// TIA Portal V17 export
// export: Created 2023-05-07T12:12:23.0932555Z, ExportSetting WithDefaults, DisplayName Totally Integrated Automation Portal, DisplayVersion V17, DisplayName TIA Portal Openness, DisplayVersion V17, DisplayName TIA Portal Version Control Interface, DisplayVersion V17, DisplayName TIA Portal Test Suite Advanced, DisplayVersion V17, DisplayName STEP 7 Professional, DisplayVersion V17, DisplayName SIMATIC Energy Suite, DisplayVersion V17, DisplayName STEP 7 Safety, DisplayVersion V17, DisplayName WinCC Professional, DisplayVersion V17
DATA_BLOCK "Measurement_DB"   // DB12
VERSION : 0.1
// stored: AutoNumber true, InstanceOfName Measurement, InstanceOfType FB
"Measurement"
   // VAR_INPUT
   //    y : Real;
   // END_VAR
   // VAR_OUTPUT
   //    r : Real;
   //    finish : Bool;
   // END_VAR
   // VAR
   //    r_array : Array[0..249] of Real;
   //    y_array : Array[0..249] of Real;
   //    i : Int;
   // END_VAR
BEGIN
END_DATA_BLOCK
